FUNCTION_BLOCK FB_SignalHandlingIntern IMPLEMENTS I_SignalHandling
VAR_INPUT
	bInputSignal					:			BOOL;					// Software intern input signal
END_VAR
VAR_OUTPUT
	bOutputSignal					:			BOOL;					// Software intern output singnal, e.g. delayed, inverted
END_VAR
VAR
	bEnableInputLocal				:			BOOL;					// Enabling processing of input signal
END_VAR

METHOD Enable
VAR_INPUT
	bEnable	: BOOL;
END_VAR
	
	bEnableInputLocal	:=		bEnable;
END_METHOD

METHOD SetOutput
	
	bOutputSignal	:=	bInputSignal AND bEnableInputLocal;
END_METHOD

END_FUNCTION_BLOCK

(* stored: Version 1.1.0.1, ProductVersion 3.1.4024.15
   POU FB_SignalHandlingIntern: Id {c35e22c0-e410-47ec-91b7-8d63ca8ef2a0}, SpecialFunc None
   Method Enable: Id {71a25948-8cf7-4d3c-add6-bbff29aecd02}
   Method SetOutput: Id {1a938916-71d0-4536-b245-b8b41d3e1530} *)
